PROGRAM PRG_LVCP1_Group1
VAR
    // Function Block Instance
    fbContactor: FB_ContactorControl;

    // Contactor 1 IO Structure  
    stContactor_IO: ST_ContactorIO;
    
    // Başlangıç konfigürasyonu için flag
    bContactorInitDone: BOOL := FALSE;
    bCapacitorInitDone: BOOL := FALSE;	
END_VAR



	M_Contactor();
	
	M_Capacitor();

METHOD M_Capacitor : BOOL
VAR
    nGroupIndex : INT;
END_VAR
	nGroupIndex := 0;  // Grup 1 için index
	
	IF NOT bCapacitorInitDone THEN
	
		// Grup 1 değerlerini ata
		GVL_LVCP1.astCompensationGroups[nGroupIndex].rPower := 25.0;
		GVL_LVCP1.astCompensationGroups[nGroupIndex].rVoltage := 450.0;
		GVL_LVCP1.astCompensationGroups[nGroupIndex].nQuantity := 10;
		GVL_LVCP1.astCompensationGroups[nGroupIndex].sTagPrefix := '+EP6-16C1';
		GVL_LVCP1.astCompensationGroups[nGroupIndex].sProductCode := 'ENT.CXD-450-25';
		
		bCapacitorInitDone := TRUE;
	END_IF
	
	// Grup 1 aktif durumu
	GVL_LVCP1.abGroupActive[nGroupIndex] := stContactor_IO.bFeedback;
	
	M_Capacitor := TRUE;
END_METHOD

METHOD M_Contactor : BOOL
VAR_INPUT
END_VAR
IF NOT bContactorInitDone THEN
    // Konfigürasyon parametreleri
    GVL_LVCP1.stGroup1_ContactorHMI.stConfig.sProjectCode := '+EP6-17K1';
    GVL_LVCP1.stGroup1_ContactorHMI.stConfig.sProductCode := 'SCH LC1G630LSEA';
    GVL_LVCP1.stGroup1_ContactorHMI.stConfig.rRatedCurrent := 630.0;
    GVL_LVCP1.stGroup1_ContactorHMI.stConfig.rRatedVoltage := 1000.0;
    GVL_LVCP1.stGroup1_ContactorHMI.stConfig.nPhaseCount := 3;
    GVL_LVCP1.stGroup1_ContactorHMI.stConfig.tFeedbackDelay := T#500MS;
    GVL_LVCP1.stGroup1_ContactorHMI.stConfig.tWeldedDelay := T#2S;
    GVL_LVCP1.stGroup1_ContactorHMI.stConfig.dwOperationLimit := 100000;
    // Başlangıç bakım sayacı
    GVL_LVCP1.stGroup1_ContactorHMI.stStatistics.dwRemainingOperations := GVL_LVCP1.stGroup1_ContactorHMI.stConfig.dwOperationLimit;
	
	bContactorInitDone := TRUE;
END_IF	
	
// Function Block Çağrısı
fbContactor(
    // Fiziksel Girişler
    bFeedback 		:= stContactor_IO.bFeedback,
    bPLCControl 	:= stContactor_IO.bPLCControl,
    
    // Güvenlik Girişleri
    bSafetyLoop 	:= GVL_Alarm.bSafetyLoop,
    bInterlock 		:= FALSE,
    
    // Sistem Girişleri
    bMasterReset 	:= GVL_Alarm.bMasterReset,
    
    // HMI Bağlantısı
    stHMI 			:= GVL_LVCP1.stGroup1_ContactorHMI,
    
    // Fiziksel Çıkış
    bOutput 		=> stContactor_IO.bOutput
);

// SQL Kayıt İşlemi
IF GVL_LVCP1.stGroup1_ContactorHMI.stStatistics.bNewOperationFlag THEN
    // SQL kayıt fonksiyonunu çağır
    GVL_LVCP1.stGroup1_ContactorHMI.stStatistics.bNewOperationFlag := FALSE;
END_IF
END_METHOD

END_PROGRAM

(* stored: Version 1.1.0.1, ProductVersion 3.1.4024.15
   POU PRG_LVCP1_Group1: Id {08f9beec-4397-4262-90ac-511b04ba46ef}, SpecialFunc None
   Method M_Capacitor: Id {f891aa9c-a6e8-40e4-86e8-657058e6ebc0}
   Method M_Contactor: Id {ddfe2ccd-3771-44fd-8a5e-24db62a5a9b2} *)
